(* Basic interface for autodocs tests. *)
INTERFACE I_Basic

METHOD Init : BOOL
VAR_INPUT
    bForce : BOOL;
END_VAR
END_METHOD

PROPERTY Ready : BOOL
GET
END_GET
END_PROPERTY

END_INTERFACE

(* stored: Version 1.1.0.1
   Itf I_Basic: Id {44444444-4444-4444-4444-444444444401}
   Method Init: Id {44444444-4444-4444-4444-444444444402}
   Property Ready: Id {44444444-4444-4444-4444-444444444403}
   Get Get: Id {44444444-4444-4444-4444-444444444404} *)
